{attribute 'enable_dynamic_creation'}
FUNCTION_BLOCK FB_Vial EXTENDS FB_UsingPiece
VAR
	pSeptum: POINTER TO FB_PieceBase;
	nTopLevel: DINT;
	nBottomLevel: DINT;
END_VAR

{attribute 'object_name' := 'FB_init'}
METHOD FB_init : BOOL
VAR_INPUT
	/// if TRUE, the retain variables are initialized (warm start / cold start)
	bInitRetains: BOOL;
	/// if TRUE, the instance afterwards gets moved into the copy code (online change)
	bInCopyCode: BOOL;
END_VAR
bUsingPiece := TRUE;
eObjectType := E_ObjectType.OBJECTTYPE_Vial;
eObjectGroup := E_ObjectGroup.OBJECTGROUP_Piece;
END_METHOD

{attribute 'object_name' := 'M_ClearAllProps'}
METHOD M_ClearAllProps

VAR_INPUT
	bIgnoreParent : BOOL; //Es wird das gesamte OD gelöscht. -> Zeiger auf Parent nicht mehr gültig!
END_VAR
pSeptum := 0;
SUPER^.M_ClearAllProps(bIgnoreParent);
END_METHOD

{attribute 'object_name' := 'M_GetAllProps'}
METHOD M_GetAllProps : ERRORID
VAR_INPUT
	refCmdData: REFERENCE TO ST_CmdData;
END_VAR
SUPER^.M_GetAllProps(refCmdData);
nCurrentPropIndex := nCurrentPropIndex + 1;
refCmdData.n32Data[nCurrentPropIndex] := nTopLevel;
nCurrentPropIndex := nCurrentPropIndex + 1;
refCmdData.n32Data[nCurrentPropIndex] := nBottomLevel;
END_METHOD

{attribute 'object_name' := 'M_SetAllProps'}
METHOD M_SetAllProps : ERRORID
VAR_INPUT
	refCmdData: REFERENCE TO ST_CmdData;
END_VAR
M_SetAllProps := SUPER^.M_SetAllProps(refCmdData);

IF M_SetAllProps > 0 THEN
	RETURN;
END_IF
nCurrentPropIndex := nCurrentPropIndex + 1;
nTopLevel := refCmdData.n32Data[nCurrentPropIndex];
nCurrentPropIndex := nCurrentPropIndex + 1;
nBottomLevel := refCmdData.n32Data[nCurrentPropIndex];
nNoOfProps := nCurrentPropIndex + 1;
END_METHOD

METHOD M_SetSingleProp : ERRORID
VAR_INPUT
	refCmdData : REFERENCE TO  ST_CmdData;
END_VAR
IF refCmdData.aHeader[1] < 13 THEN	//Property-Nr
	M_SetSingleProp := SUPER^.M_SetSingleProp(refCmdData);
ELSE
	IF refCmdData.aHeader[1] = 13 THEN
		//bIsOpen := DINT_TO_BOOL(refCmdData.n32Data[0]);
		;
	ELSIF refCmdData.aHeader[1] = 14 THEN
		nTopLevel := refCmdData.n32Data[0];
	ELSIF refCmdData.aHeader[1] = 15 THEN
		nBottomLevel := refCmdData.n32Data[0];
	ELSE
		M_SetSingleProp := E_ErrorIdCmd.ERRORID_InvalidProperty;
	END_IF
END_IF
END_METHOD

PROPERTY P_nBottomLevel : DINT
GET
P_nBottomLevel := nBottomLevel;
END_GET
END_PROPERTY

PROPERTY P_nTopLevel : DINT
GET
P_nTopLevel := nTopLevel;
END_GET
END_PROPERTY

PROPERTY P_pLatestChild : POINTER TO FB_PieceBase
GET
IF pSeptum > 0 THEN
	P_pLatestChild := pSeptum;	
ELSE
	P_pLatestChild := THIS;
END_IF
END_GET
END_PROPERTY

PROPERTY P_pSeptum : POINTER TO FB_PieceBase
GET
P_pSeptum := pSeptum;
END_GET
SET
pSeptum := P_pSeptum;
END_SET
END_PROPERTY

END_FUNCTION_BLOCK

(* stored: Version 1.1.0.1, ProductVersion 3.1.4022.18
   POU FB_Vial: Id {e56e79ad-755c-47a3-9f91-0926d60671f2}, SpecialFunc None
   Method FB_init: Id {dc97a6db-7594-483c-b952-6a1eda0dd441}
   Method M_ClearAllProps: Id {c636e6b6-e625-46af-8128-b85da5c4536b}
   Method M_GetAllProps: Id {bd305124-dda6-430d-9680-0b6957e4a5b4}
   Method M_SetAllProps: Id {c71150f0-c274-4f3f-91c1-0e607b552a52}
   Method M_SetSingleProp: Id {18146b88-1129-4fba-a15a-877c50f6527c}
   Property P_nBottomLevel: Id {88f66479-b16d-4d9d-b7aa-98a765631393}
   Get Get: Id {a17ff1e0-ac5c-471e-964b-4f318d191cc1}
   Property P_nTopLevel: Id {d9e11507-9e94-4c4a-80a7-10f28a2e8391}
   Get Get: Id {6a87a6aa-64e2-4c59-8dad-81cb2256513d}
   Property P_pLatestChild: Id {79b2169c-f70b-48d7-907d-f5ddb16ed16a}
   Get Get: Id {e61f3d0b-589d-48e7-91d2-f9e9d5dff586}
   Property P_pSeptum: Id {ccb33d7d-d1ba-438d-9119-e6a1d89acb62}
   Get Get: Id {a3eb10f1-de5c-4142-902a-38389423bfda}
   Set Set: Id {22135a4d-04af-4944-ab0c-fe0ecf876106} *)
